TYPE TFMachinePalletizer_CoordinateApprendimento :
STRUCT
	X : TFMachinePalletizer_LatoApprendimento;
	Y : TFMachinePalletizer_LatoApprendimento;
	Z : TFMachinePalletizer_LatoApprendimento;
	J : TFMachinePalletizer_LatoApprendimento;
END_STRUCT
END_TYPE

(* stored: Version 1.1.0.1, ProductVersion 3.1.4024.11
   DUT TFMachinePalletizer_CoordinateApprendimento: Id {a7b85eee-a307-4f27-92a6-c6945778521b} *)
